{attribute 'linkalways'} 
{attribute 'no_explicit_call' := 'This FB is a CLASS and must be accessed using methods or properties'}
{attribute 'enable_dynamic_creation'}
FUNCTION_BLOCK Node_F_VN_CheckFunctionInitialization EXTENDS VisionNode
VAR
    eFunction : _ETcVnInitializableFunction(ETcVnInitializableFunction.TCVN_IF_OCR);
    nOptions : _ULINT(0);
    hrPrev : _HRESULT(S_OK);
	hresult : _HRESULT(S_OK);
END_VAR

METHOD PUBLIC  Clone : I_Node
VAR
	pNode : POINTER TO Node_F_VN_CheckFunctionInitialization;
END_VAR
pNode := __NEW(Node_F_VN_CheckFunctionInitialization);
Clone := pNode^;
END_METHOD

METHOD FB_init : BOOL
VAR_INPUT
	bInitRetains : BOOL; // if TRUE, the retain variables are initialized (warm start / cold start)
	bInCopyCode : BOOL;  // if TRUE, the instance afterwards gets moved into the copy code (online change)
END_VAR
AddParameter('eFunction', eFunction);
AddInput('nOptions', nOptions);
AddInput('hrPrev', hrPrev);
AddOutput('hresult',hresult);
END_METHOD

METHOD PROTECTED OnExecute
hresult.Value := F_VN_CheckFunctionInitialization(
	eFunction := eFunction.Value,
    nOptions := nOptions.Value,
	hrPrev:= hrPrev.Value);
END_METHOD

METHOD PUBLIC PreExecutionCheck
VAR_INPUT
	Check : I_PreExecutionChecks;
END_VAR
END_METHOD

END_FUNCTION_BLOCK

(* stored: Version 1.1.0.1, ProductVersion 3.1.4024.13
   POU Node_F_VN_CheckFunctionInitialization: Id {a35b728f-f110-0477-375a-2a190912ca41}, SpecialFunc None
   Folder Constructor: Id {6936bd6b-31b2-07fa-3988-f184c4de9811}
   Method Clone: Id {957877c0-7b09-0abb-1027-eaf2d1714e4c}
   Method FB_init: Id {ec7bb0bc-db95-0e6f-3fc6-13c2d888a36d}
   Method OnExecute: Id {68bf8a03-1eec-090d-1fbb-1b5d7327e875}
   Method PreExecutionCheck: Id {6a70babf-88cf-0893-2b52-201237efdfa5} *)
